(* CoDeSys 2.3.8.0 project: Laser_G67HP_3.pro *)
(* Libraries: STANDARD.LIB 5.6.98 12:03:02, TcBase.lib 6.6.06 16:41:28, TcSystem.lib 9.3.07 18:11:38, TcSystemCX.lib 5.3.07 17:55:46, TcUtilities.lib 29.3.07 15:04:14 *)

(* Global variable list: Globale_Variablen *)
VAR_GLOBAL

	(* Hardwareeingänge *)
	INot_Aus 			 	AT %IX0.0 : BOOL; (* Eingang 1 *)
	IDruckW			  	AT %IX0.1 : BOOL; (* Eingang 2 *)
	ISchututuer	  		AT %IX0.2 : BOOL; (* Eingang 3 *)
	ISchutzhaube  		AT %IX0.3 : BOOL; (* Eingang 4 *)
	IHWT_EIN			 	AT %IX0.4 : BOOL; (* Eingang 5 *)
	IHWT_AUS			AT %IX0.5 : BOOL; (* Eingang 6 *)
	IHWT_Quitt  			AT %IX0.6 : BOOL; (* Eingang 7 *)
	IRES1					AT %IX0.7 : BOOL; (* Eingang 8 *)

       IINI_Ueberlast  		AT %IX1.0 : BOOL; (* Eingang 9 *)
	IINI_IndexVor	  		AT %IX1.1 : BOOL; (* Eingang 10 *)
	IINI_IndexRueck  		AT %IX1.2 : BOOL; (* Eingang 11 *)
	IINI_Kupplung  		AT %IX1.3 : BOOL; (* Eingang 12 *)
	IINI_SpeicherZu		AT %IX1.4 : BOOL; (* Eingang 13 *)
	IRES3		 			AT %IX1.5 : BOOL; (* Eingang 14 *)
	IRES4					AT %IX1.6 : BOOL;
	IRES5		 			AT %IX1.7 : BOOL;

	IKammError  			AT %IX2.0 : BOOL; (* Eingang 17 *)
	IKammEnable  		AT %IX2.1 : BOOL; (* Eingang 18 *)
	IKammOutput  		AT %IX2.2 : BOOL; (* Eingang 19 *)
	IRES6		 			AT %IX2.3 : BOOL; (* Eingang 20 *)
	IAbsaug100P 			AT %IX2.4 : BOOL; (* Eingang 21 *)
	IAbsaugFilter			AT %IX2.5 : BOOL; (* Eingang 22 *)
	IRES					AT %IX2.6 : BOOL; (* Eingang 23 *)
	IFU_BB				AT %IX2.7 : BOOL; (* Eingang 24 *)

	IFrgMoma1 			AT %IX3.0 : BOOL;
	IFrgMoma2 			AT %IX3.1 : BOOL;
	ShutterZu	 			AT %IX3.2 : BOOL;
	ShutterAuf	 			AT %IX3.3 : BOOL;
	ILAS_HWFehler		AT %IX3.4 : BOOL;
	ILAS_SWIO 			AT %IX3.5 : BOOL;
	ILAS_Redy	 		AT %IX3.6 : BOOL;
	ILAS_AuftragEnde 	AT %IX3.7 : BOOL;

	ILasDataBit0 			AT %IX4.0 : BOOL;
	ILasDataBit1 	 		AT %IX4.1 : BOOL;
	ILasDataBit2 		 	AT %IX4.2 : BOOL;
	ILasDataBit3 		 	AT %IX4.3 : BOOL;
	ILasDataBit4 	 		AT %IX4.4 : BOOL;
	ILasDataBit5 	 		AT %IX4.5 : BOOL;
	ILasResI1	 		 	AT %IX4.6 : BOOL;
	ILasResI2 			 AT %IX4.7 : BOOL;

	(*Eingänge für die Panel Tasten*)

	IAPosKS1Input  		AT%IW20:INT;	 	(*Speicher 1 Füllstand analoger Eingang*)
	IARES1				AT%IW22:INT;
	IASSIDgInput			 AT %ID44:UDINT;	(* Drehgeber *)


	QHAmpelGn		 	AT %QX0.0 : BOOL; (* Ventil Pneumatik  *)
	QHAmpelRt	  		AT %QX0.1 : BOOL; (* Ausgang 2 *)
	QHAmpelGb 			AT %QX0.2 : BOOL; (* Ausgang 3 *)
	QRES1				AT %QX0.3 : BOOL; (* Ausgang 4 *)
	QHTasteEin			AT %QX0.4 : BOOL; (* Ausgang 5 *)
	QHTasteAus			AT %QX0.5 : BOOL; (* Ausgang 6 *)
	QHTasteQuitt			AT %QX0.6 : BOOL; (* Ausgang 7 *)
	QRES2				AT %QX0.7 : BOOL; (* Ausgang 8 *)

	QLasMark				AT %QX1.0 : BOOL; (* Ausgang 9 *)
	QLasMarkstop		AT %QX1.1 : BOOL; (* Ausgang 10 *)
	QLasProg1			AT %QX1.2 : BOOL; (* Ausgang 11 *)
	QLasProg2			AT %QX1.3 : BOOL; (* Ausgang 12 *)
	QLasRes2			AT %QX1.4 : BOOL; (* Ausgang 13 *)
	QLasRes3			AT %QX1.5 : BOOL; (* Ausgang 14 *)
	QFrgNaechst			AT %QX1.6 : BOOL; (* Ausgang 15 *)
	QAntriebeEin		     	AT %QX1.7 : BOOL; (* Ausgang 16 *)

	QMotVor	 			AT %QX2.0 : BOOL; (* Ausgang 9 *)
	QMotRueck			AT %QX2.1 : BOOL; (* Ausgang 10 *)
	QSaugAnford			AT %QX2.2 : BOOL; (* Ausgang 11 *)
	QVIndex				AT %QX2.3 : BOOL; (* Ausgang 12 *)
	QVUeberlast			AT %QX2.4 : BOOL; (* Ausgang 13 *)
	QVHaupt				AT %QX2.5 : BOOL; (* Ausgang 14 *)
	QVASpeicher			AT %QX2.6 : BOOL; (* Ausgang 15 *)
	QKammTrigg			AT %QX2.7 : BOOL; (* Ausgang 16 *)

	QASollwMot			AT%QW4:WORD; (*Ausgangswort 1*)
	QARes				 	AT%QW6:WORD; (*Ausgangswort 2*)

(* Anfang der Variablen für Kopmunikation SPS <> Visu *)
	TP_LaserAktiv	:			BOOL:= TRUE;
	TP_LaserHand:			BOOL;
	TP_RefSetzen:			BOOL;
	TP_KammeraAktiv:		BOOL:=TRUE;
	TP_MVor:					BOOL;
	TP_Mrueck:				BOOL;
	TP_MVorS:				BOOL;
	TP_MrueckS:				BOOL;

	TP_Hand:					BOOL;
	TP_Auto:					BOOL;
	TP_ZNullen:				BOOL;
	TPTypIndex:				WORD;
	TPTypSpeichern:			BOOL;
	TPKettenTyp: 				ARRAY[0..3] OF WORD;

	S_StUeberlast:			BOOL;
	S_StLaser:				BOOL;
	S_StKammera:			BOOL;
	S_StKupplung	:			BOOL;
	S_StSpeicherSchutz:		BOOL;
	S_StLaserSchutz:			BOOL;
	S_StSpeicher:				BOOL;
	S_StSammelstoerung:	BOOL;
	S_StDruck:				BOOL;
	S_StNotAus:				BOOL;
	S_StRef:					BOOL;
	S_StSchutzTuer:			BOOL;
	S_StSchutzhaube: 		BOOL;
	S_StAbsaugFilter:			BOOL;	(*Absauger Filter NIO*)
	S_StAbsaug100p:			BOOL;	(*Störung Absauger*)
	S_StShutter:				BOOL;

	S_StLasAuftragEnde:		BOOL;	(* Auftrag Ende*)
	S_StLasShutterZu:			BOOL;	(* Shutter zu *)
	S_StLasSoftware:			BOOL;	(*Software NIO*)
	S_StLasHardware:		BOOL;	(*Hardware NIO*)
	S_StIndexVor:			BOOL;	(*Index vor NIO*)
	S_StIndexRueck:			BOOL;	(*Index rueck NIO*)

	S_MSpeicherVoll:			BOOL;
	S_MShutterBetrieb:		BOOL;
	S_MSpeicherLeer:		BOOL;
	S_MWarteSpeicher:		BOOL;
	S_MHand:					BOOL;
	S_FKamera:				BOOL;
	S_FLaser:					BOOL;
	S_MAutoStart:				BOOL;
	S_MAutoStop:				BOOL;
	SI_Gliederzahl:			INT;
	SI_ProgNr:				INT;
	SI_FPosLaser:			INT;  (*wird nicht genutzt*)
	SI_FPosKamera:			INT;  (*wird nicht genutzt*)
	SKettenTyp:ARRAY[0..3] OF WORD;
(* ENDE*)

	Skal_IC_SSI_DG_Input: 	DINT;
	Skal_SSI_DG_4:			DINT;
	ZeigerReg:				INT;
	ZeigerKette: 				WORD;
	ImpulsPos: 				BOOL;
	ImpulsNeg: 				BOOL;
	Sammelstoerung: BOOL;

	V_Erster_Zyklus: BOOL;
	REF_IO: BOOL;
	AktTypIndexAlt: WORD;
	AktTypindex:WORD;
	NextTypIndex:WORD;
	PosErreicht: BOOL;


	NextTypIndexAlt: WORD;
	A_wechsell: BOOL;
	S1_AutoStop: BOOL;
	S2_Posstart: BOOL;
	S3_POSStop: BOOL;
	S4_IndexVor: BOOL;
	S5_LaserStart: BOOL;
	S6_IndexRueck: BOOL;

	Stoerunganlage:WORD;

	Zeiger_LMKontrolle: INT;
	FNichtMarkiert: BOOL;

	AktTypOL: BOOL;
	S_FrgEinzug: BOOL;
	KSEnIn: BOOL;
	KSEnOut: BOOL;
	TON_IIndexVor: TON;
	Stufe1: INT;
END_VAR

VAR_GLOBAL RETAIN



	(*Hinterlegte Kettentypen 64 Kettentypen 0-63  , 0=>Gliederzahl, 1-3=>Positionen der ersten bis dritten Außenlasche zum Lasern*)
	(*KettenTyp[x,2]=0 Bedeutet keine zweite Laserung an einer Kette*)
	(*KettenTyp[x,3]=0 Bedeutet keine dritte Laserung an einer Kette*)
	(*KettenTyp[x,1]=0 Nullter Kettentyp keine Laserung*)
	(*KettenTyp[x,0]=0 Ungültiger Eintrag *)

	(*Beispiel für eine Kette: 124 Glieder mit einer Laserung an der ersten Außenlasche gespeichert als Typ 5*)
	(*KettenTyp[5,0]=124   Kettentyp[5,1]=1 Kettentyp[5,2]=0  Kettentyp[5,3]=0*)
	KettenTyp							AT%QW100:ARRAY [0..63,0..3] OF WORD;

	(* Einträge in das Register RegMarkierung:
		X.0=1   Trennstelle
		X.1=1   Lasersollstelle, 
		X.2=1   Rückmeldung von Laser gelasert, 
		X.3=1   Fehler keine Rückmeldung von Laser "Gelesert"
		X.4=1   Rückmeldung Kammera Laserstelle
		X.5=1	Fehler keine Rückmeldung von Kammera "Laserstelle"
*)
	RegMarkierung					AT%QB1000:ARRAY[1..500] OF BYTE;


(*   Fehlerzähler für die erste Seite. Fehler können ohne Password zurückgesetzt werden*)

	SI_FKamera				AT%QW70:INT;
	SI_FLaser 				AT%QW72:INT;
	SI_IO						AT%QW74:INT;
	SI_NIO 					AT%QW76:INT;
(*	ZeigerGlied				AT%QW304:INT;				(* Zeiger für die Glieder in der Anlage zeigt auf das Glied unter der Trennstelle *)
	ZeigerAchtelGlied			AT%QW306:INT;
*)
END_VAR

(* Data type *)
TYPE DriveControl :
STRUCT
	ManOn: BOOL := FALSE; (* Visu -> SPS: Antrieb ein (nur bei FU-Antrieben) *)
	ManOff: BOOL := FALSE; (* Visu -> SPS: Antrieb aus (nur bei FU-Antrieben) *)
	ManFwd: BOOL := FALSE; (* Visu -> SPS: Antrieb im Handbetrieb langsam vorwärts *)
	ManBwd: BOOL := FALSE; (* Visu -> SPS: Antrieb im Handbetrieb langsam rückwärts *)
	TeilungVor: BOOL := FALSE; (* Visu -> SPS: Kette um eine Teilung vor (nur bei Servo-Antrieben) *)
	TeilungZur: BOOL := FALSE; (* Visu -> SPS: Kette um eine Teilung zurück (nur bei Servo-Antrieben) *)
	EnManCtrl: BOOL := FALSE; (* SPS -> Visu: Freigabe manuelle Steuerung *)
	ActOn: BOOL := FALSE; (* SPS -> Visu: Antrieb eingeschaltet *)
	ActOff: BOOL := FALSE; (* SPS -> Visu: Antrieb ausgeschaltet *)
	Error: BOOL := FALSE; (* SPS -> Visu: Störung Antrieb *)
END_STRUCT
END_TYPE

(* Data type *)
TYPE KettenTyp :
STRUCT
	PF: ARRAY [0..19] OF UDINT := 0,410,819,1229,1638,2048,2458,2867,3277,3686,4049,4506,4915,5328,5734,6144,6554,6963,7373,7782;

END_STRUCT
END_TYPE

(* Data type *)
TYPE KS_Control :
STRUCT
	EnInput: BOOL := FALSE; (* Freigabe Befüllen *)
	EnOutput: BOOL := FALSE; (* Freigabe Entleeren *)
	ActState: INT := 0; (* aktueller zustand für Visu *)
END_STRUCT
END_TYPE

(* Data type *)
TYPE KS_Control_1 :
STRUCT
	EnInput: BOOL := FALSE; (* Freigabe Befüllen *)
	EnOutput: BOOL := FALSE; (* Freigabe Entleeren *)
	ActState: INT := 0; (* aktueller zustand für Visu *)
END_STRUCT
END_TYPE

(* Data type *)
TYPE MotorControl :
STRUCT
	ManOn: BOOL := FALSE; (* Visu -> SPS: Antrieb im Handbetrieb ein *)
	ManOff: BOOL := FALSE; (* Visu -> SPS: Antrieb im Handbetrieb aus *)
	EnManCtrl: BOOL := FALSE; (* SPS -> Visu: Freigabe manuelle Steuerung *)
	ActOn: BOOL := FALSE; (* SPS -> Visu: Antrieb eingeschaltet *)
	ActOff: BOOL := FALSE; (* SPS -> Visu: Antrieb ausgeschaltet *)
	Error: BOOL := FALSE; (* SPS -> Visu: Störung Antrieb *)
END_STRUCT
END_TYPE

(* Data type *)
TYPE PneumControl :
STRUCT
	SetOn: BOOL := FALSE; (* Visu -> SPS: Arbeitsstellung anfahren *)
	SetOff: BOOL := FALSE; (* Visu -> SPS: Grundstellung anfahren *)
	EnSet: BOOL := FALSE; (* SPS -> Visu: Freigabe manuell Steuerung *)
	ActOn: BOOL := FALSE; (* SPS -> Visu: Zylinder in Arbeitsstellung *)
	ActOff: BOOL := FALSE; (* SPS -> Visu: Zylinder in Grundstellung *)
	Error: BOOL := FALSE; (* SPS -> Visu: Störung Zylinder oder Endschalter *)
END_STRUCT
END_TYPE

(* Data type *)
TYPE PosControl :
STRUCT
	PosSet: INT := 0; (* Positionssollwert [mm] *)
	ActPos: INT := 0; (* Positionsistwert [mm] *)
	PosLimitLo: INT := 0; (* unterer Grenzwert Sollposition [mm] *)
	PosLimitHi: INT := 0; (* oberer Grenzwert Sollposition [mm] *)
	StartPos: BOOL := FALSE; (* Visu -> SPS: Positionierung starten *)
	StoppPos: BOOL := FALSE; (* Visu -> SPS: Positionierung abbrechen *)
	ManPosUp: BOOL := FALSE; (* Visu -> SPS: Handbetrieb Positon erhöhen *)
	ManPosDn: BOOL := FALSE; (* Visu -> SPS: Handbetrieb Positon verringern *)
	EnPosSet: BOOL := FALSE; (* SPS -> Visu: Freigabe Sollwerteingabe *)
	EnManPos: BOOL := FALSE; (* SPS -> Visu: Freigabe manuelle Positionierung *)
	ActOn: BOOL := FALSE; (* SPS -> Visu: Antrieb eingeschaltet *)
	ActOff: BOOL := FALSE; (* SPS -> Visu: Antrieb ausgeschaltet *)
	Error: BOOL := FALSE; (* SPS -> Visu: Störung Antrieb *)
END_STRUCT
END_TYPE

(* Data type *)
TYPE StationControl :
STRUCT
	StepCounter: INT; (* SPS -> Visu: Schrittzähler *)
	SingleStep: BOOL := FALSE; (* Visu -> SPS: Einzelschritt weiterschalten *)
	SingleCycle: BOOL := FALSE; (* Visu -> SPS: Einzelzyklus ausführen *)
	StartCycle: BOOL := FALSE; (* Zyklus im Auto-Betrieb starten *)
	ManInit: BOOL := FALSE; (* Visu -> SPS: Grundstellung anfahren *)
	AutoInit: BOOL := FALSE; (* Grundstellung im Auto-Betrieb anfahren *)
	SetFinished: BOOL := FALSE; (* Visu -> SPS: Fertigmeldung setzen *)
	WaitPos: BOOL := FALSE; (* Station in Warteposition für Stopp *)
	EnSemiAutoCtrl: BOOL := FALSE; (* SPS -> Visu: Steuerung Halbautomatikbetrieb freigeben; Freigabe für SingleStep, SingleCycle, InitPos und SetFinished *)
	InitPos: BOOL := FALSE; (* Station in Grundstellung *)
	Finished: BOOL := FALSE; (* Station fertig *)
	ErrorInitPos: BOOL := FALSE; (* Störung Grundstellung nicht erreicht *)
	ErrorCycleTime: BOOL := FALSE; (* Störung Zeitüberschreitung Zyklus *)
	ActState: INT := 0; (* SPS -> Visu: Zustand der Station: 0 = Störung, 1 = bereit, 2 = aktiv *)
END_STRUCT
END_TYPE

(* POU INIT, ST *)
PROGRAM INIT

VAR

END_VAR
(* Der Kettentyp wird von Laserrechner ausgewählt *)
NextTypIndex.0:=ILasDataBit0;
NextTypIndex.1:=ILasDataBit1;
NextTypIndex.2:=ILasDataBit2;
NextTypIndex.3:=ILasDataBit3;
NextTypIndex.4:=ILasDataBit4;
NextTypIndex.5:=ILasDataBit5;



(*  Wenn NuxtTypIndex = 0 dann Auftrag ohne Laserung *)
(* Wenn Laser per Touchpannel deaktiviert dann auch Auftrag ohne Laserung *)
IF TP_LaserAktiv = FALSE THEN
	NextTypIndex:=0;
END_IF

(* Wenn Wechsell von Auftrag ohne Laserung auf Auftrag mit Laserung dann Referenz nue anfordern *)

IF	AktTypIndex = 0 AND NextTypIndex <> 0 THEN
	REF_IO:=FALSE;
END_IF




(* Wenn die Maschine eingeschaltet wird ist eine Ref Fahrt durchzuführen *)
IF V_Erster_Zyklus=FALSE THEN
	REF_IO:=FALSE;
	AktTypIndex:=NextTypIndex;
END_IF
V_Erster_Zyklus:=TRUE;



(* Trennstelle der Kette auf Indexposition fahren und Referenzieren *)
IF (*REF_IO= FALSE AND*) TP_RefSetzen= TRUE THEN
	ZeigerKette:=KettenTyp[AktTypIndex,0];
	REF_IO:=TRUE;
END_IF


(* Wenn Kettentyp gewechselt wurde muß Auftragswechsellbitt gesetzt werden *)
IF NextTypIndex <> NextTypIndexAlt THEN
	A_wechsell:=TRUE;
END_IF
NextTypIndexAlt:=NextTypIndex;

(* Der Auftragswechsell wird durchgeführt wenn das Ende der  Kette von Alten Auftrag unter der Leserstelle gelangt *)
(* Auftragswechsellbit wird auf FALSE gesetzt *)
IF   ZeigerKette = KettenTyp[AktTypIndex,0] THEN
	AktTypIndex:=NextTypIndex;
	SI_ProgNr:=AktTypIndex;
	SI_Gliederzahl:= KettenTyp[AktTypIndex,0];
	A_wechsell:=FALSE;
	ZeigerKette := KettenTyp[AktTypIndex,0];
END_IF

IF	NextTypIndex = 63 THEN
	SI_ProgNr:=63;
END_IF

IF	ImpulsPos =TRUE THEN
	(*Alten Eintrag im Register Löschen*)
	(*Laser wird dann die Markierung eintragen*)
	RegMarkierung[ZeigerReg]:=0;

	(*Trennstell in das Register eintragen*)
	IF   ZeigerKette = KettenTyp[AktTypIndex,0] THEN
	RegMarkierung[ZeigerReg].0:=TRUE;
	END_IF

END_IF
END_PROGRAM

(* POU MAIN_1, FBD *)
PROGRAM MAIN_1
VAR
	SollPos1: SollPos;
	ASMSollW1: AsmSollW;
	Motorsteuerung1: Motorsteuerun;
	Betriebsarten1: Betriebsarten;
	Kettenspeicher1: Kettenspeicher;

	Saugersteuerung1: Saugersteuerung;
	Kettentypen1: Kettentypen;
	Indexsteuerung1: Indexsteuernung;
	Anlagenstoerung1: Anlagestoerung;
	Lasersteuerung1: Lasersteuerung;
	LaserMeldungKontrolle1: LaserMeldungKontrolle;
	Kammera1: Kammera;
	FK1: BOOL;
	V1: BOOL;
	PF1: R_TRIG;
	TP1: TP;
END_VAR
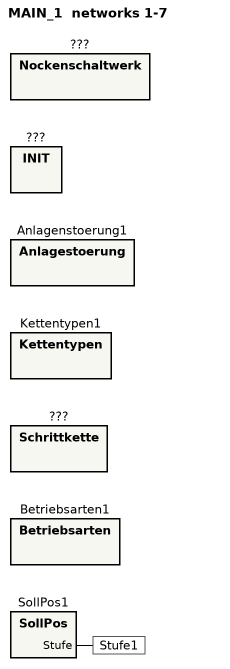
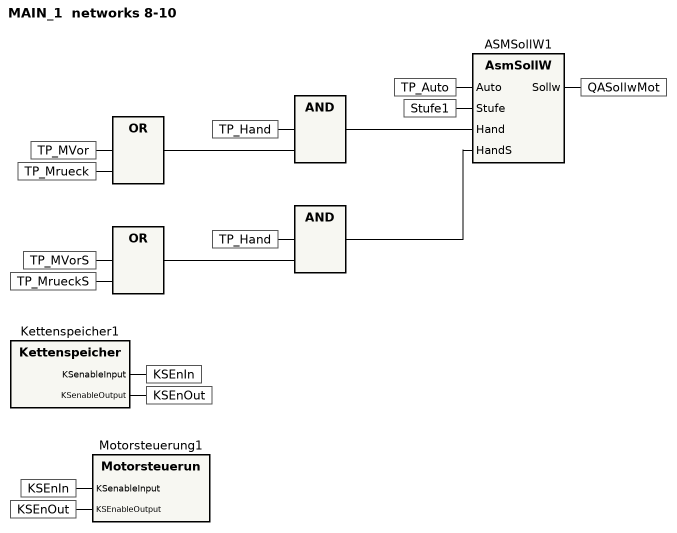
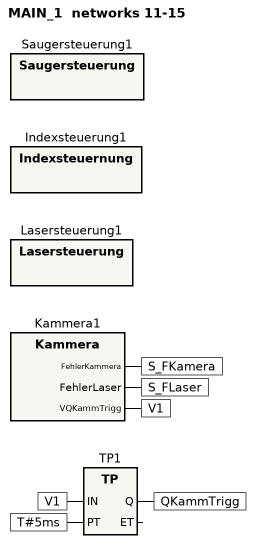
_FBD_ (* Function Block Diagram *)
NETWORK 1
	???:Nockenschaltwerk()
NETWORK 2
	???:INIT()
NETWORK 3
	Anlagenstoerung1:Anlagestoerung()
NETWORK 4
	Kettentypen1:Kettentypen()
NETWORK 5
	???:Schrittkette()
NETWORK 6
	Betriebsarten1:Betriebsarten()
NETWORK 7
	SollPos1:SollPos() => Stufe1
NETWORK 8
	ASMSollW1:AsmSollW(Auto: TP_Auto, Stufe: Stufe1, Hand: AND(TP_Hand, OR(TP_MVor, TP_Mrueck)), HandS: AND(TP_Hand, OR(TP_MVorS, TP_MrueckS))) => QASollwMot
NETWORK 9
	Kettenspeicher1:Kettenspeicher(KSenableOutput => KSEnOut) => KSEnIn
NETWORK 10
	Motorsteuerung1:Motorsteuerun(KSenableInput: KSEnIn, KSEnableOutput: KSEnOut)
NETWORK 11
	Saugersteuerung1:Saugersteuerung()
NETWORK 12
	Indexsteuerung1:Indexsteuernung()
NETWORK 13
	Lasersteuerung1:Lasersteuerung()
NETWORK 14
	Kammera1:Kammera(FehlerLaser => S_FLaser, VQKammTrigg => V1) => S_FKamera
NETWORK 15
	TP1:TP(IN: V1, PT: T#5ms) => QKammTrigg
_END_FBD_
(* the same logic as Structured Text *)
(* Network 1: see the listing above *)
(* Network 2: see the listing above *)
(* Network 3 *)
Anlagenstoerung1();
(* Network 4 *)
Kettentypen1();
(* Network 5: see the listing above *)
(* Network 6 *)
Betriebsarten1();
(* Network 7 *)
SollPos1();
Stufe1 := SollPos1.Stufe;
(* Network 8 *)
ASMSollW1(Auto := TP_Auto, Stufe := Stufe1, Hand := TP_Hand AND (TP_MVor OR TP_Mrueck), HandS := TP_Hand AND (TP_MVorS OR TP_MrueckS));
QASollwMot := ASMSollW1.Sollw;
(* Network 9 *)
Kettenspeicher1();
KSEnOut := Kettenspeicher1.KSenableOutput;
KSEnIn := Kettenspeicher1.KSenableInput;
(* Network 10 *)
Motorsteuerung1(KSenableInput := KSEnIn, KSEnableOutput := KSEnOut);
(* Network 11 *)
Saugersteuerung1();
(* Network 12 *)
Indexsteuerung1();
(* Network 13 *)
Lasersteuerung1();
(* Network 14 *)
Kammera1();
S_FLaser := Kammera1.FehlerLaser;
V1 := Kammera1.VQKammTrigg;
S_FKamera := Kammera1.FehlerKammera;
(* Network 15 *)
TP1(IN := V1, PT := T#5ms);
QKammTrigg := TP1.Q;
END_PROGRAM

(* POU Funktionsbausteine/SollPos, ST *)
FUNCTION_BLOCK SollPos
VAR_INPUT
END_VAR
VAR_OUTPUT
	Stufe: INT := 1;
END_VAR
VAR
	ZeigerStufe1: INT;
	ZeigerStufe2: INT;
	ZeigerStufe3: INT;
	ZeigerStufe4: INT;
	ZeigerStufe5: INT;

END_VAR
(* Wenn Referenz gesetzt oder wurde oder nach dem Einschalten erst langsam anfahren *)

IF TP_RefSetzen= TRUE OR V_Erster_Zyklus= FALSE THEN
	Stufe:=1;
END_IF

 TP_RefSetzen:= FALSE;


IF	ImpulsPos =TRUE THEN


	(* Geschwindigkeitsstufen für die Positionierung ermitteln *)
	(* Zeiger für die Stufen berechnen *)
	(* Bearbeitung nur wenn Aussenlasche*)
	IF ZeigerKette.0=FALSE THEN
		ZeigerStufe1:=ZeigerKette+2;
		IF ZeigerStufe1>KettenTyp[AktTypindex,0] THEN
			ZeigerStufe1:=ZeigerStufe1-KettenTyp[AktTypindex,0];
		END_IF
		ZeigerStufe2:=ZeigerStufe1+2;
		IF ZeigerStufe2>KettenTyp[AktTypindex,0] THEN
			ZeigerStufe2:=ZeigerStufe2-KettenTyp[AktTypindex,0];
		END_IF
		ZeigerStufe3:=ZeigerStufe2+2;
		IF ZeigerStufe3>KettenTyp[AktTypindex,0] THEN
			ZeigerStufe3:=ZeigerStufe3-KettenTyp[AktTypindex,0];
		END_IF
		ZeigerStufe4:=ZeigerStufe3+2;
		IF ZeigerStufe4>KettenTyp[AktTypindex,0] THEN
			ZeigerStufe4:=ZeigerStufe4-KettenTyp[AktTypindex,0];
		END_IF
		ZeigerStufe5:=ZeigerStufe4+2;
		IF ZeigerStufe5>KettenTyp[AktTypindex,0] THEN
			ZeigerStufe5:=ZeigerStufe5-KettenTyp[AktTypindex,0];
		END_IF




		(* In Abhängikeit von der Entfernung der nächsten Lasche welche gelesert werden soll wird die Geschwindigkeit des Motors in 6 Stufen geregelt*)
		(* Wenn Auftragswechsell anliegt wird die Geschwindigkeit des Motors verringert bisdas Ende der alten Kette die Laserungsstelle erreicht*)
		(* Sollgeschwindigkeit ist auf Stufe 6 eingestellt. Wenn die Laserungsstelle auf fünfte Aussenlasche vor Laserungsstelle ist dann langsamer auf Stufe 5*)

		IF ZeigerStufe5 = KettenTyp[AktTypindex,1]*2 OR ZeigerStufe5 = KettenTyp[AktTypindex,2]*2 OR ZeigerStufe5 = KettenTyp[AktTypindex,3]*2THEN
			Stufe:=5;
		ELSE
			Stufe:=6;
		END_IF
		(* Wenn Auftragswechsell und Kettenende von alten Auftrag auf 5 Außenlasche vor Laserungsstelle dan auf Stufe 5 stellen*)
		IF	A_wechsell = TRUE AND (ZeigerKette+10) = KettenTyp[AktTypindex,0] THEN
			Stufe:=5;
		END_IF


		(* Wenn die Laserungsstelle auf vierte Aussenlasche vor Laserungsstelle ist dann langsamer auf Stufe 4*)
		IF ZeigerStufe4 = KettenTyp[AktTypindex,1]*2 OR ZeigerStufe4 = KettenTyp[AktTypindex,2]*2 OR ZeigerStufe4 = KettenTyp[AktTypindex,3]*2THEN
			Stufe:=4;
		END_IF
		(* Wenn Auftragswechsell und Kettenende von alten Auftrag auf 4 Außenlasche vor Laserungsstelle dan auf Stufe 4 stellen*)
		IF	A_wechsell = TRUE AND (ZeigerKette+8) = KettenTyp[AktTypindex,0] THEN
			Stufe:=4;
		END_IF



		IF ZeigerStufe3 = KettenTyp[AktTypindex,1]*2 OR ZeigerStufe3 = KettenTyp[AktTypindex,2]*2 OR ZeigerStufe3 = KettenTyp[AktTypindex,3]*2THEN
			Stufe:=3;
		END_IF
		(* Wenn Auftragswechsell und Kettenende von alten Auftrag auf 3 Außenlasche vor Laserungsstelle dan auf Stufe 3 stellen*)
		IF	A_wechsell = TRUE AND (ZeigerKette+6) = KettenTyp[AktTypindex,0] THEN
			Stufe:=3;
		END_IF



		IF ZeigerStufe2 = KettenTyp[AktTypindex,1]*2 OR ZeigerStufe2 = KettenTyp[AktTypindex,2]*2 OR ZeigerStufe2 = KettenTyp[AktTypindex,3]*2THEN
			Stufe:=2;
		END_IF
		(* Wenn Auftragswechsell und Kettenende von alten Auftrag auf 2 Außenlasche vor Laserungsstelle dan auf Stufe 2 stellen*)
		IF	A_wechsell = TRUE AND (ZeigerKette+4) = KettenTyp[AktTypindex,0] THEN
			Stufe:=2;
		END_IF

		IF ZeigerStufe1 = KettenTyp[AktTypindex,1]*2 OR ZeigerStufe1 = KettenTyp[AktTypindex,2]*2 OR ZeigerStufe1 = KettenTyp[AktTypindex,3]*2THEN
			Stufe:=1;
		END_IF
		(* Wenn Auftragswechsell und Kettenende von alten Auftrag auf 1 Außenlasche vor Laserungsstelle dan auf Stufe 1 stellen*)
		IF	A_wechsell = TRUE AND (ZeigerKette+2) = KettenTyp[AktTypindex,0] THEN
			Stufe:=1;
		END_IF

		(* Position erreicht melden und Laserungssollstelle in das Register Schreiben *)
		IF ZeigerKette = KettenTyp[AktTypindex,1]*2 OR ZeigerKette = KettenTyp[AktTypindex,2]*2 OR ZeigerKette = KettenTyp[AktTypindex,3]*2THEN
			IF RegMarkierung[ZeigerReg].2 = FALSE THEN
				PosErreicht:=TRUE;
				RegMarkierung[ZeigerReg].1:=TRUE;
			END_IF
		END_IF
	END_IF


	(*  Bearbeitung nur bei Innenlasche an der Laserstelle *)
	(*  Wenn die Lasersollposition überfahren ohne zu lasern dann  PosErreicht zurücksetzen *)
	IF ZeigerKette.0=TRUE  THEN
	PosErreicht:=FALSE;
	END_IF

END_IF
END_FUNCTION_BLOCK

(* POU Funktionsbausteine/AsmSollW, ST *)
FUNCTION_BLOCK AsmSollW
VAR

END_VAR

VAR_INPUT
	Auto: BOOL;
	Stufe: INT;
	Hand: BOOL;
	HandS:BOOL;
END_VAR
VAR_OUTPUT
	Sollw: INT;
END_VAR
IF  Auto = TRUE THEN
	IF Stufe= 6 THEN
	Sollw:=30000;
	END_IF
	IF Stufe= 5 THEN
	Sollw:=27000;
	END_IF
	IF Stufe= 4 THEN
	Sollw:=18000;
	END_IF
	IF Stufe= 3 THEN
	Sollw:=15000;
	END_IF
	IF Stufe= 2 THEN
	Sollw:=10000;
	END_IF
	IF Stufe= 1 THEN
	Sollw:=1000;
	END_IF
END_IF

IF	Hand=TRUE  THEN
	Sollw:=5000;
END_IF


IF	HandS=TRUE  THEN
	Sollw:=15000;
END_IF
END_FUNCTION_BLOCK

(* POU Funktionsbausteine/Motorsteuerun, FBD *)
FUNCTION_BLOCK Motorsteuerun
VAR_INPUT
	KSenableInput: BOOL;
	KSEnableOutput: BOOL;
END_VAR
VAR_OUTPUT
END_VAR
VAR
	PF_AutoStart: R_TRIG;
	PF_AutoStop: R_TRIG;
	StopGoMot: RS;
END_VAR
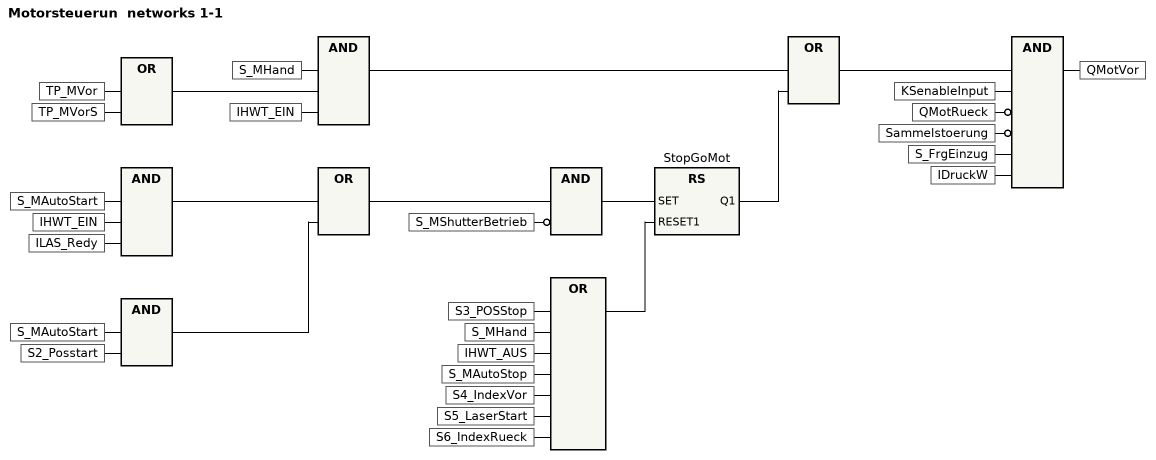
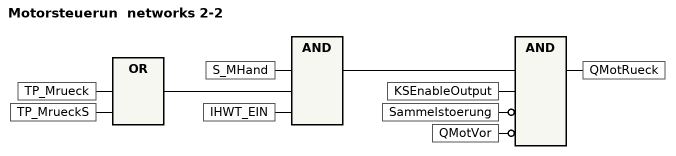
_FBD_ (* Function Block Diagram *)
NETWORK 1 (* Ansteuerung des Motors M1 in Positive richtung *)
	AND(OR(AND(S_MHand, OR(TP_MVor, TP_MVorS), IHWT_EIN), StopGoMot:RS(SET: AND(OR(AND(S_MAutoStart, IHWT_EIN, ILAS_Redy), AND(S_MAutoStart, S2_Posstart)), NOT S_MShutterBetrieb), RESET1: OR(S3_POSStop, S_MHand, IHWT_AUS, S_MAutoStop, S4_IndexVor, S5_LaserStart, S6_IndexRueck))), KSenableInput, NOT QMotRueck, NOT Sammelstoerung, S_FrgEinzug, IDruckW) => QMotVor
NETWORK 2 (* Ansteuerung Motor M1 in negative Richtung *)
	AND(AND(S_MHand, OR(TP_Mrueck, TP_MrueckS), IHWT_EIN), KSEnableOutput, NOT Sammelstoerung, NOT QMotVor) => QMotRueck
_END_FBD_
(* the same logic as Structured Text *)
(* Network 1: Ansteuerung des Motors M1 in Positive richtung *)
StopGoMot(SET := ((S_MAutoStart AND IHWT_EIN AND ILAS_Redy) OR (S_MAutoStart AND S2_Posstart)) AND NOT S_MShutterBetrieb, RESET1 := S3_POSStop OR S_MHand OR IHWT_AUS OR S_MAutoStop OR S4_IndexVor OR S5_LaserStart OR S6_IndexRueck);
QMotVor := ((S_MHand AND (TP_MVor OR TP_MVorS) AND IHWT_EIN) OR StopGoMot.Q1) AND KSenableInput AND NOT QMotRueck AND NOT Sammelstoerung AND S_FrgEinzug AND IDruckW;
(* Network 2: Ansteuerung Motor M1 in negative Richtung *)
QMotRueck := (S_MHand AND (TP_Mrueck OR TP_MrueckS) AND IHWT_EIN) AND KSEnableOutput AND NOT Sammelstoerung AND NOT QMotVor;
END_FUNCTION_BLOCK

(* POU Funktionsbausteine/Betriebsarten, FBD *)
FUNCTION_BLOCK Betriebsarten
VAR_INPUT
END_VAR
VAR_OUTPUT
END_VAR
VAR
	Blink_TON1: TON;
	Blink_TON2: TON;
	VIHWT_AUS: BOOL;
END_VAR
VAR (* helpers for the ST form of the networks *)
	_p1 : BOOL;
	_p2 : BOOL;
END_VAR
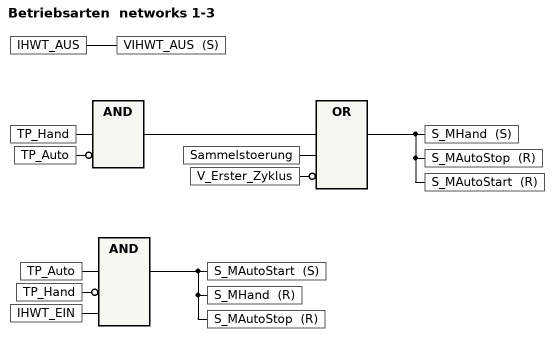
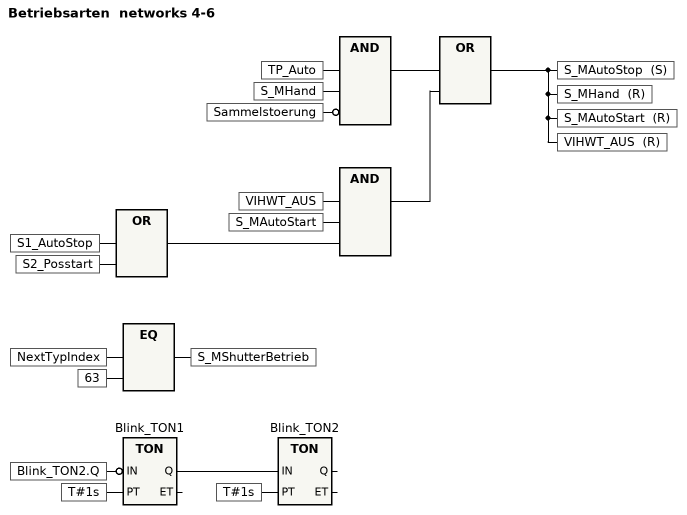
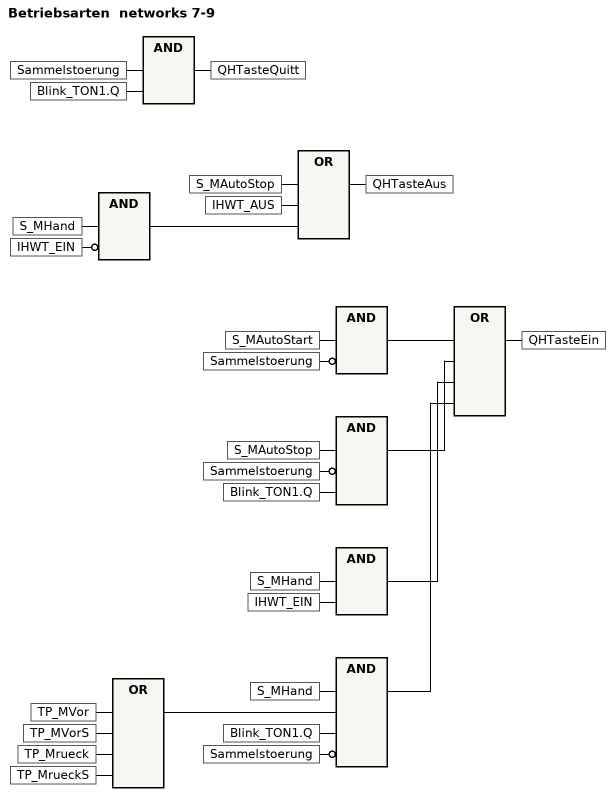
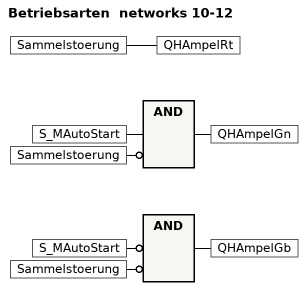
_FBD_ (* Function Block Diagram *)
NETWORK 1
	IHWT_AUS => S VIHWT_AUS
NETWORK 2
	OR(AND(TP_Hand, NOT TP_Auto), Sammelstoerung, NOT V_Erster_Zyklus) => S S_MHand, R S_MAutoStop, R S_MAutoStart
NETWORK 3
	AND(TP_Auto, NOT TP_Hand, IHWT_EIN) => S S_MAutoStart, R S_MHand, R S_MAutoStop
NETWORK 4
	OR(AND(TP_Auto, S_MHand, NOT Sammelstoerung), AND(VIHWT_AUS, S_MAutoStart, OR(S1_AutoStop, S2_Posstart))) => S S_MAutoStop, R S_MHand, R S_MAutoStart, R VIHWT_AUS
NETWORK 5
	EQ(NextTypIndex, 63) => S_MShutterBetrieb
NETWORK 6
	Blink_TON2:TON(IN: Blink_TON1:TON(IN: NOT Blink_TON2.Q, PT: T#1s), PT: T#1s)
NETWORK 7
	AND(Sammelstoerung, Blink_TON1.Q) => QHTasteQuitt
NETWORK 8
	OR(S_MAutoStop, IHWT_AUS, AND(S_MHand, NOT IHWT_EIN)) => QHTasteAus
NETWORK 9
	OR(AND(S_MAutoStart, NOT Sammelstoerung), AND(S_MAutoStop, NOT Sammelstoerung, Blink_TON1.Q), AND(S_MHand, IHWT_EIN), AND(S_MHand, OR(TP_MVor, TP_MVorS, TP_Mrueck, TP_MrueckS), Blink_TON1.Q, NOT Sammelstoerung)) => QHTasteEin
NETWORK 10
	Sammelstoerung => QHAmpelRt
NETWORK 11
	AND(S_MAutoStart, NOT Sammelstoerung) => QHAmpelGn
NETWORK 12
	AND(NOT S_MAutoStart, NOT Sammelstoerung) => QHAmpelGb
_END_FBD_
(* the same logic as Structured Text *)
(* Network 1 *)
IF IHWT_AUS THEN VIHWT_AUS := TRUE; END_IF;
(* Network 2 *)
_p1 := (TP_Hand AND NOT TP_Auto) OR Sammelstoerung OR NOT V_Erster_Zyklus;
IF _p1 THEN S_MHand := TRUE; S_MAutoStop := FALSE; S_MAutoStart := FALSE; END_IF;
(* Network 3 *)
IF TP_Auto AND NOT TP_Hand AND IHWT_EIN THEN S_MAutoStart := TRUE; S_MHand := FALSE; S_MAutoStop := FALSE; END_IF;
(* Network 4 *)
_p2 := (TP_Auto AND S_MHand AND NOT Sammelstoerung) OR (VIHWT_AUS AND S_MAutoStart AND (S1_AutoStop OR S2_Posstart));
IF _p2 THEN S_MAutoStop := TRUE; S_MHand := FALSE; S_MAutoStart := FALSE; VIHWT_AUS := FALSE; END_IF;
(* Network 5 *)
S_MShutterBetrieb := NextTypIndex = 63;
(* Network 6 *)
Blink_TON1(IN := NOT Blink_TON2.Q, PT := T#1s);
Blink_TON2(IN := Blink_TON1.Q, PT := T#1s);
(* Network 7 *)
QHTasteQuitt := Sammelstoerung AND Blink_TON1.Q;
(* Network 8 *)
QHTasteAus := S_MAutoStop OR IHWT_AUS OR (S_MHand AND NOT IHWT_EIN);
(* Network 9 *)
QHTasteEin := (S_MAutoStart AND NOT Sammelstoerung) OR (S_MAutoStop AND NOT Sammelstoerung AND Blink_TON1.Q) OR (S_MHand AND IHWT_EIN) OR (S_MHand AND (TP_MVor OR TP_MVorS OR TP_Mrueck OR TP_MrueckS) AND Blink_TON1.Q AND NOT Sammelstoerung);
(* Network 10 *)
QHAmpelRt := Sammelstoerung;
(* Network 11 *)
QHAmpelGn := S_MAutoStart AND NOT Sammelstoerung;
(* Network 12 *)
QHAmpelGb := NOT S_MAutoStart AND NOT Sammelstoerung;
END_FUNCTION_BLOCK

(* POU Funktionsbausteine/Kettenspeicher, FBD *)
FUNCTION_BLOCK Kettenspeicher
VAR_INPUT
END_VAR
VAR_OUTPUT
	KSenableInput: BOOL;
	KSenableOutput: BOOL;
END_VAR
VAR
	RS1: RS;
END_VAR
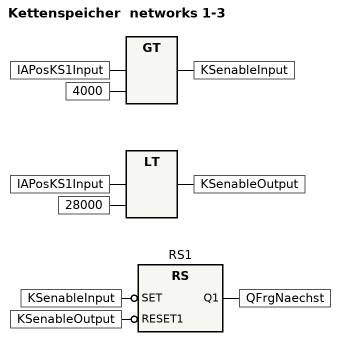
_FBD_ (* Function Block Diagram *)
NETWORK 1
	GT(IAPosKS1Input, 4000) => KSenableInput
NETWORK 2
	LT(IAPosKS1Input, 28000) => KSenableOutput
NETWORK 3
	RS1:RS(SET: NOT KSenableInput, RESET1: NOT KSenableOutput) => QFrgNaechst
_END_FBD_
(* the same logic as Structured Text *)
(* Network 1 *)
KSenableInput := IAPosKS1Input > 4000;
(* Network 2 *)
KSenableOutput := IAPosKS1Input < 28000;
(* Network 3 *)
RS1(SET := NOT KSenableInput, RESET1 := NOT KSenableOutput);
QFrgNaechst := RS1.Q1;
END_FUNCTION_BLOCK

(* POU Funktionsbausteine/Saugersteuerung, FBD *)
FUNCTION_BLOCK Saugersteuerung
VAR_INPUT
END_VAR
VAR_OUTPUT
END_VAR
VAR
	TON1: TON;
	TOF1: TOF;
END_VAR
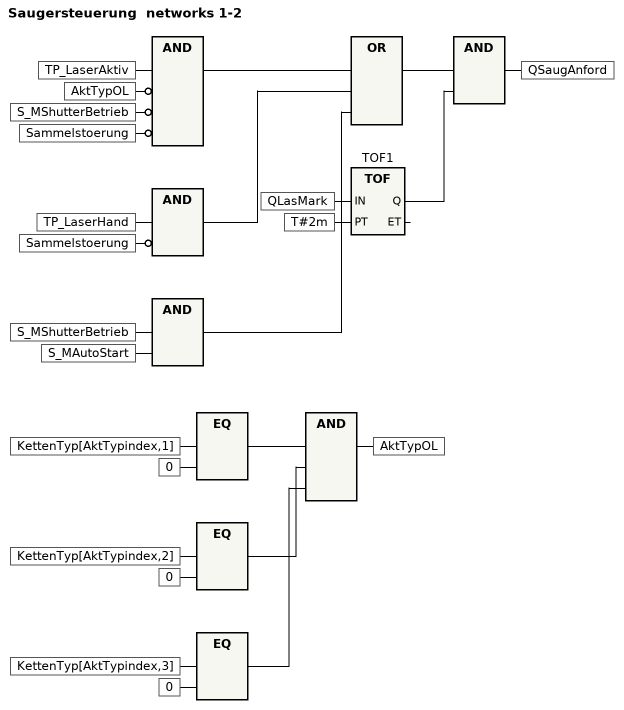
_FBD_ (* Function Block Diagram *)
NETWORK 1
	AND(OR(AND(TP_LaserAktiv, NOT AktTypOL, NOT S_MShutterBetrieb, NOT Sammelstoerung), AND(TP_LaserHand, NOT Sammelstoerung), AND(S_MShutterBetrieb, S_MAutoStart)), TOF1:TOF(IN: QLasMark, PT: T#2m)) => QSaugAnford
NETWORK 2
	AND(EQ(KettenTyp[AktTypindex,1], 0), EQ(KettenTyp[AktTypindex,2], 0), EQ(KettenTyp[AktTypindex,3], 0)) => AktTypOL
_END_FBD_
(* the same logic as Structured Text *)
(* Network 1 *)
TOF1(IN := QLasMark, PT := T#2m);
QSaugAnford := ((TP_LaserAktiv AND NOT AktTypOL AND NOT S_MShutterBetrieb AND NOT Sammelstoerung) OR (TP_LaserHand AND NOT Sammelstoerung) OR (S_MShutterBetrieb AND S_MAutoStart)) AND TOF1.Q;
(* Network 2 *)
AktTypOL := ((KettenTyp[AktTypindex,1]) = 0) AND ((KettenTyp[AktTypindex,2]) = 0) AND ((KettenTyp[AktTypindex,3]) = 0);
END_FUNCTION_BLOCK

(* POU Funktionsbausteine/Kettentypen, ST *)
FUNCTION_BLOCK Kettentypen
VAR_INPUT
END_VAR
VAR_OUTPUT
END_VAR
VAR
END_VAR
(*  Angewählten Kettentyp für Visu bereitstellen *)

SKettenTyp[0]:=KettenTyp[TPTypIndex,0];
SKettenTyp[1]:=KettenTyp[TPTypIndex,1];
SKettenTyp[2]:=KettenTyp[TPTypIndex,2];
SKettenTyp[3]:=KettenTyp[TPTypIndex,3];


(* Editierte Kettentypen remanent speichern *)
IF TPTypSpeichern = TRUE THEN
	KettenTyp[TPTypIndex,0]:=TPKettenTyp[0];
	KettenTyp[TPTypIndex,1]:=TPKettenTyp[1];
	KettenTyp[TPTypIndex,2]:=TPKettenTyp[2];
	KettenTyp[TPTypIndex,3]:=TPKettenTyp[3];
END_IF

TPTypSpeichern:= FALSE;
END_FUNCTION_BLOCK

(* POU Funktionsbausteine/Indexsteuernung, FBD *)
FUNCTION_BLOCK Indexsteuernung
VAR_INPUT
END_VAR
VAR_OUTPUT
END_VAR
VAR
	SR1: RS;
	PF_1: R_TRIG;
	PF2: R_TRIG;
	PF_3: R_TRIG;
	PF_4: R_TRIG;
	PF_5: R_TRIG;
END_VAR
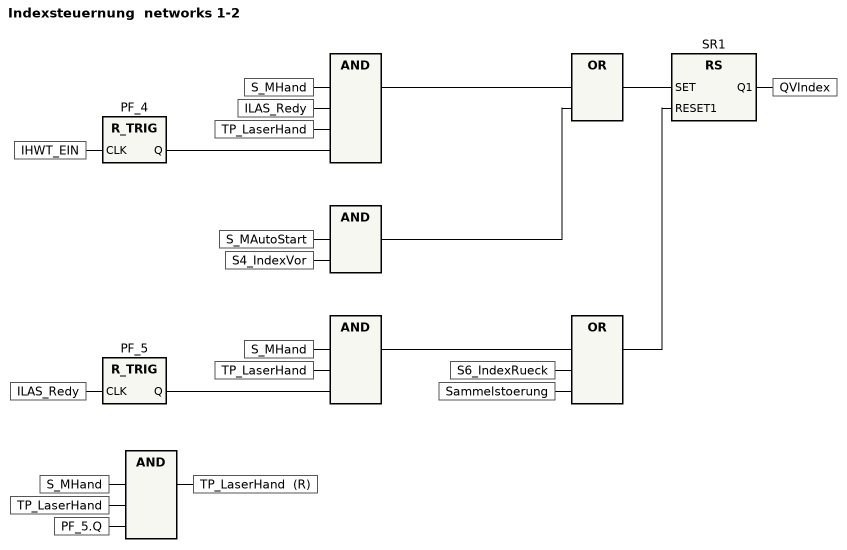
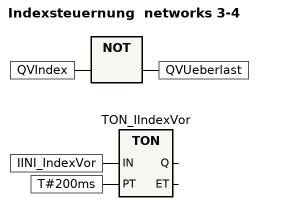
_FBD_ (* Function Block Diagram *)
NETWORK 1
	SR1:RS(SET: OR(AND(S_MHand, ILAS_Redy, TP_LaserHand, PF_4:R_TRIG(CLK: IHWT_EIN)), AND(S_MAutoStart, S4_IndexVor)), RESET1: OR(AND(S_MHand, TP_LaserHand, PF_5:R_TRIG(CLK: ILAS_Redy)), S6_IndexRueck, Sammelstoerung)) => QVIndex
NETWORK 2
	AND(S_MHand, TP_LaserHand, PF_5.Q) => R TP_LaserHand
NETWORK 3
	NOT QVIndex => QVUeberlast
NETWORK 4
	TON_IIndexVor:TON(IN: IINI_IndexVor, PT: T#200ms)
_END_FBD_
(* the same logic as Structured Text *)
(* Network 1 *)
PF_4(CLK := IHWT_EIN);
PF_5(CLK := ILAS_Redy);
SR1(SET := (S_MHand AND ILAS_Redy AND TP_LaserHand AND PF_4.Q) OR (S_MAutoStart AND S4_IndexVor), RESET1 := (S_MHand AND TP_LaserHand AND PF_5.Q) OR S6_IndexRueck OR Sammelstoerung);
QVIndex := SR1.Q1;
(* Network 2 *)
IF S_MHand AND TP_LaserHand AND PF_5.Q THEN TP_LaserHand := FALSE; END_IF;
(* Network 3 *)
QVUeberlast := NOT QVIndex;
(* Network 4 *)
TON_IIndexVor(IN := IINI_IndexVor, PT := T#200ms);
END_FUNCTION_BLOCK

(* POU Funktionsbausteine/Anlagestoerung, FBD *)
FUNCTION_BLOCK Anlagestoerung
VAR_INPUT
END_VAR
VAR_OUTPUT
END_VAR
VAR

	TON1: TON;
	PF_1: R_TRIG;
	TOF1: TOF;
	TON2: TON;
	TON3: TON;
	TON4: TON;
END_VAR
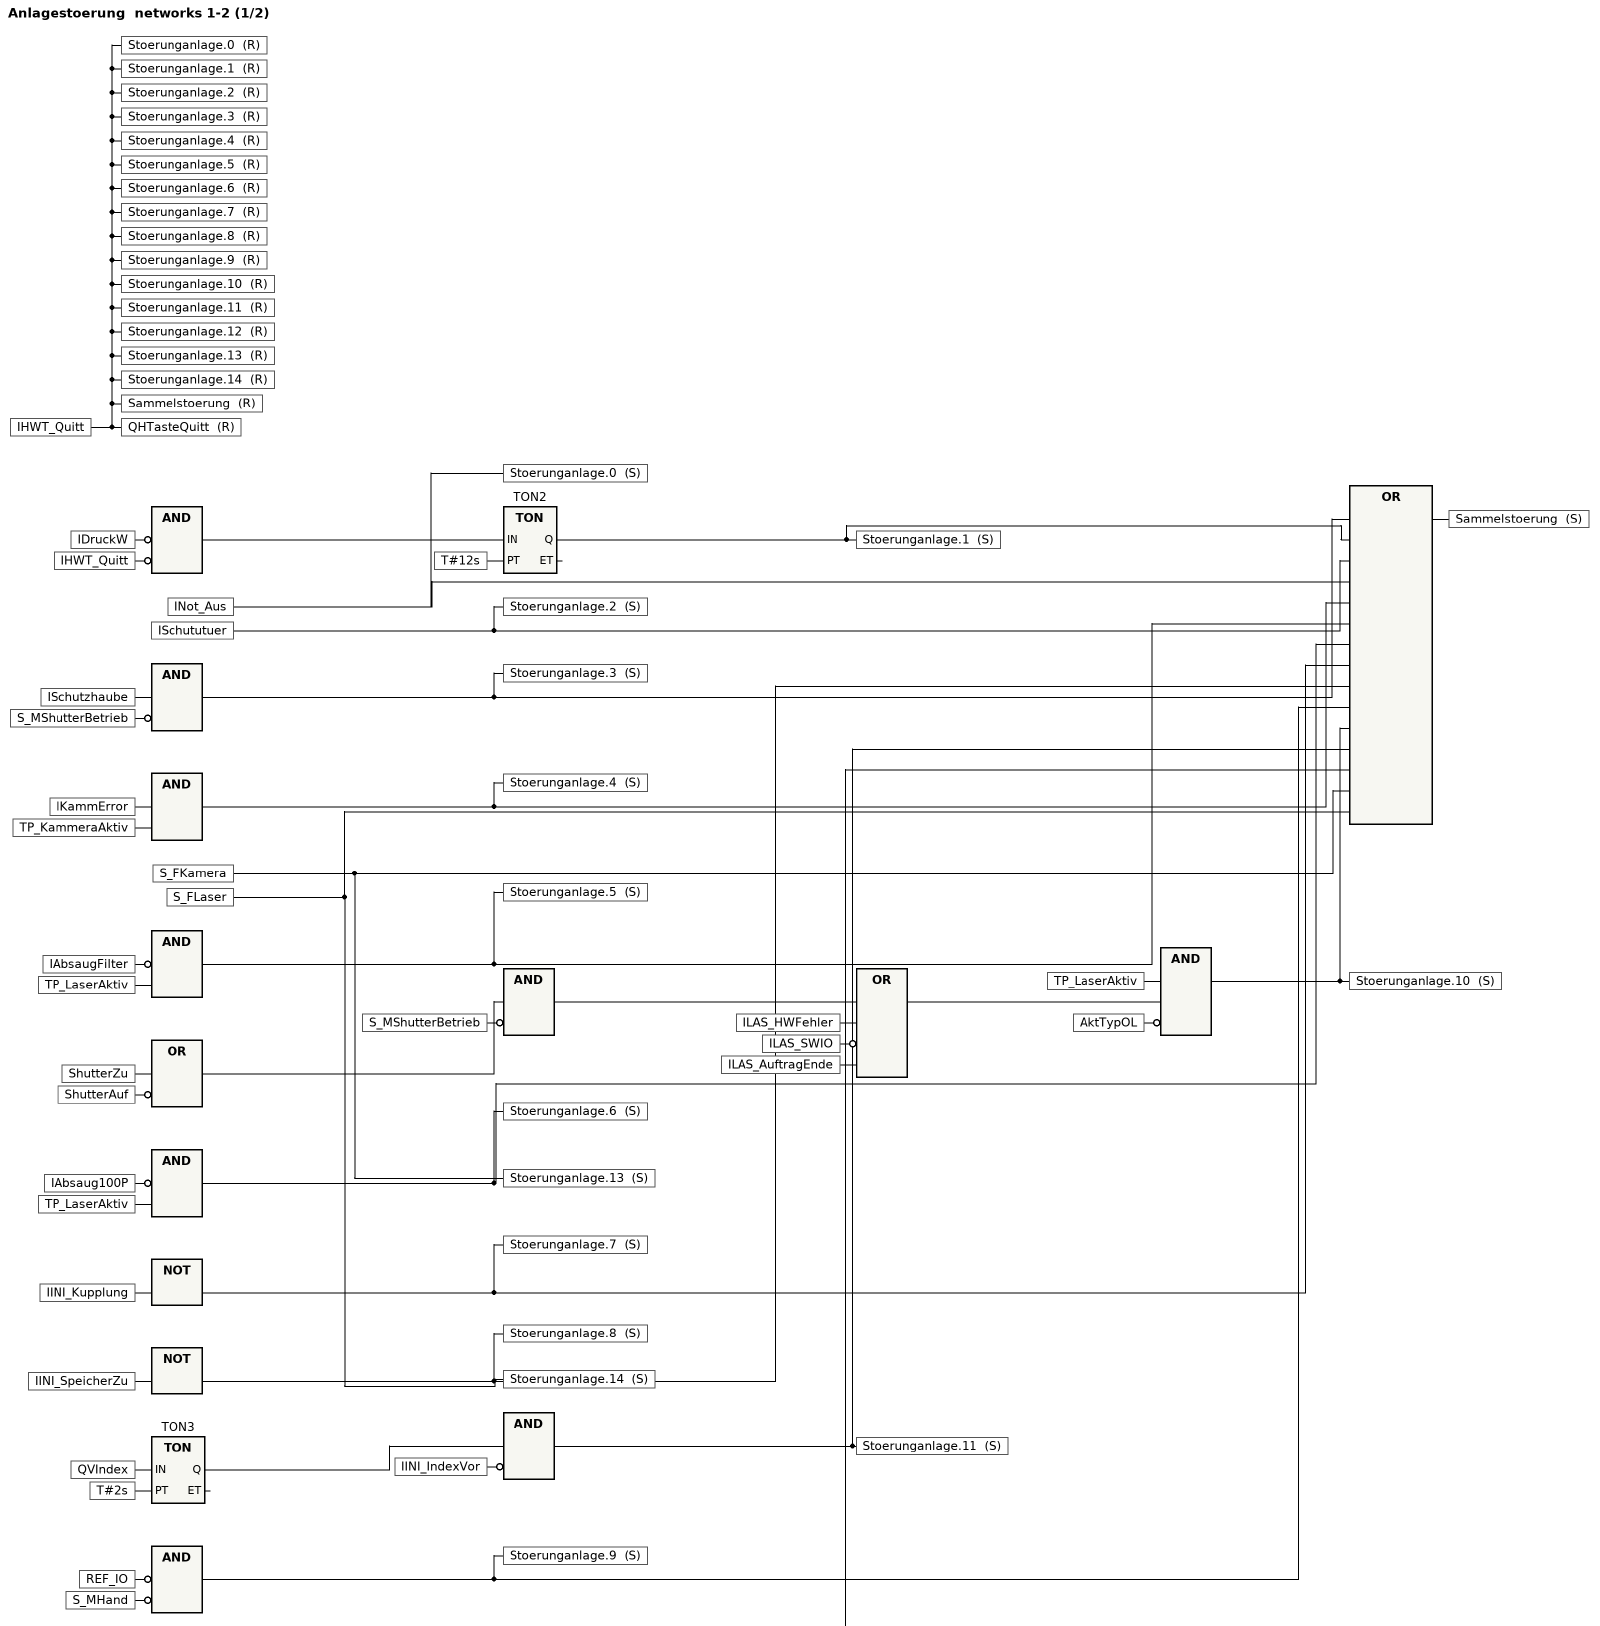
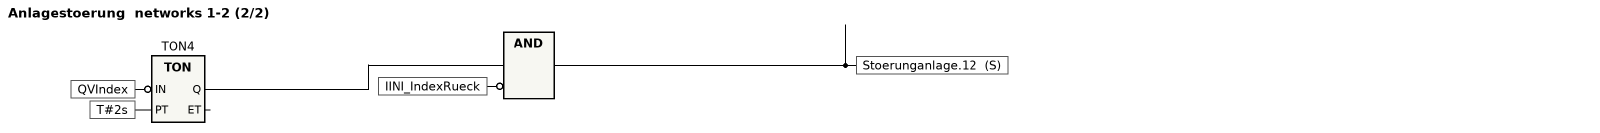
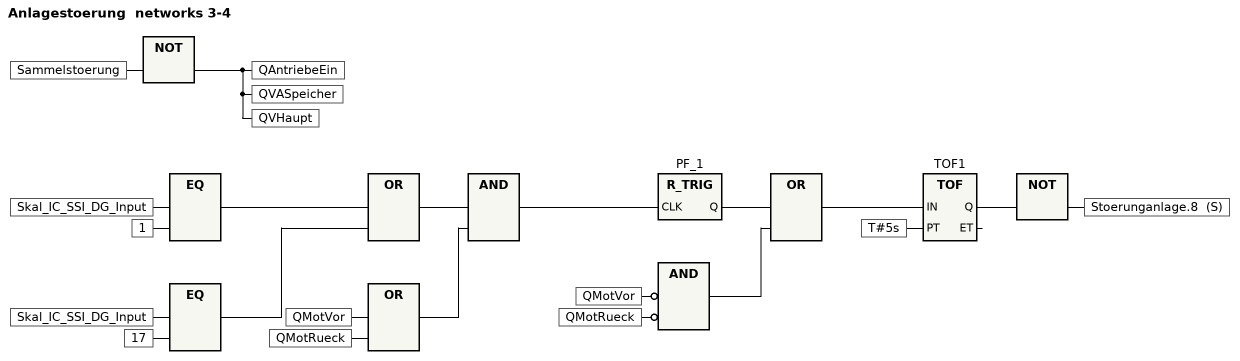
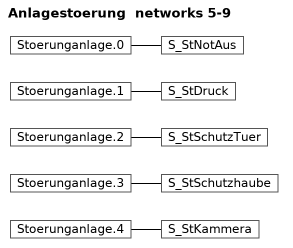
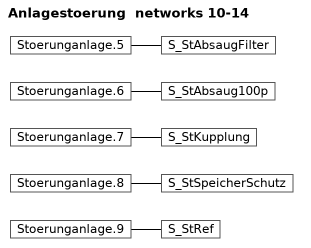
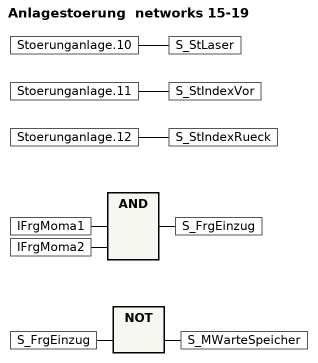
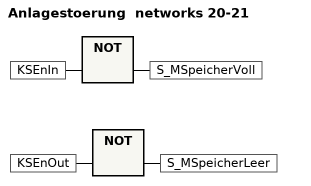
_FBD_ (* Function Block Diagram *)
NETWORK 1
	IHWT_Quitt => R Stoerunganlage.0, R Stoerunganlage.1, R Stoerunganlage.2, R Stoerunganlage.3, R Stoerunganlage.4, R Stoerunganlage.5, R Stoerunganlage.6, R Stoerunganlage.7, R Stoerunganlage.8, R Stoerunganlage.9, R Stoerunganlage.10, R Stoerunganlage.11, R Stoerunganlage.12, R Stoerunganlage.13, R Stoerunganlage.14, R Sammelstoerung, R QHTasteQuitt
NETWORK 2
	OR(<INot_Aus => S Stoerunganlage.0>, <TON2:TON(IN: AND(NOT IDruckW, NOT IHWT_Quitt), PT: T#12s) => S Stoerunganlage.1>, <ISchututuer => S Stoerunganlage.2>, <AND(ISchutzhaube, NOT S_MShutterBetrieb) => S Stoerunganlage.3>, <AND(IKammError, TP_KammeraAktiv) => S Stoerunganlage.4>, <AND(NOT IAbsaugFilter, TP_LaserAktiv) => S Stoerunganlage.5>, <AND(NOT IAbsaug100P, TP_LaserAktiv) => S Stoerunganlage.6>, <NOT IINI_Kupplung => S Stoerunganlage.7>, <NOT IINI_SpeicherZu => S Stoerunganlage.8>, <AND(NOT REF_IO, NOT S_MHand) => S Stoerunganlage.9>, <AND(TP_LaserAktiv, OR(AND(OR(ShutterZu, NOT ShutterAuf), NOT S_MShutterBetrieb), ILAS_HWFehler, NOT ILAS_SWIO, ILAS_AuftragEnde), NOT AktTypOL) => S Stoerunganlage.10>, <AND(TON3:TON(IN: QVIndex, PT: T#2s), NOT IINI_IndexVor) => S Stoerunganlage.11>, <AND(TON4:TON(IN: NOT QVIndex, PT: T#2s), NOT IINI_IndexRueck) => S Stoerunganlage.12>, <S_FKamera => S Stoerunganlage.13>, <S_FLaser => S Stoerunganlage.14>) => S Sammelstoerung
NETWORK 3
	NOT Sammelstoerung => QAntriebeEin, QVASpeicher, QVHaupt
NETWORK 4
	NOT(TOF1:TOF(IN: OR(PF_1:R_TRIG(CLK: AND(OR(EQ(Skal_IC_SSI_DG_Input, 1), EQ(Skal_IC_SSI_DG_Input, 17)), OR(QMotVor, QMotRueck))), AND(NOT QMotVor, NOT QMotRueck)), PT: T#5s)) => S Stoerunganlage.8
NETWORK 5
	Stoerunganlage.0 => S_StNotAus
NETWORK 6
	Stoerunganlage.1 => S_StDruck
NETWORK 7
	Stoerunganlage.2 => S_StSchutzTuer
NETWORK 8
	Stoerunganlage.3 => S_StSchutzhaube
NETWORK 9
	Stoerunganlage.4 => S_StKammera
NETWORK 10
	Stoerunganlage.5 => S_StAbsaugFilter
NETWORK 11
	Stoerunganlage.6 => S_StAbsaug100p
NETWORK 12
	Stoerunganlage.7 => S_StKupplung
NETWORK 13
	Stoerunganlage.8 => S_StSpeicherSchutz
NETWORK 14
	Stoerunganlage.9 => S_StRef
NETWORK 15
	Stoerunganlage.10 => S_StLaser
NETWORK 16
	Stoerunganlage.11 => S_StIndexVor
NETWORK 17
	Stoerunganlage.12 => S_StIndexRueck
NETWORK 18
	AND(IFrgMoma1, IFrgMoma2) => S_FrgEinzug
NETWORK 19
	NOT S_FrgEinzug => S_MWarteSpeicher
NETWORK 20
	NOT KSEnIn => S_MSpeicherVoll
NETWORK 21
	NOT KSEnOut => S_MSpeicherLeer
_END_FBD_
(* the same logic as Structured Text *)
(* Network 1 *)
IF IHWT_Quitt THEN Stoerunganlage.0 := FALSE; Stoerunganlage.1 := FALSE; Stoerunganlage.2 := FALSE; Stoerunganlage.3 := FALSE; Stoerunganlage.4 := FALSE; Stoerunganlage.5 := FALSE; Stoerunganlage.6 := FALSE; Stoerunganlage.7 := FALSE; Stoerunganlage.8 := FALSE; Stoerunganlage.9 := FALSE; Stoerunganlage.10 := FALSE; Stoerunganlage.11 := FALSE; Stoerunganlage.12 := FALSE; Stoerunganlage.13 := FALSE; Stoerunganlage.14 := FALSE; Sammelstoerung := FALSE; QHTasteQuitt := FALSE; END_IF;
(* Network 2 *)
IF INot_Aus THEN Stoerunganlage.0 := TRUE; END_IF;
TON2(IN := NOT IDruckW AND NOT IHWT_Quitt, PT := T#12s);
IF TON2.Q THEN Stoerunganlage.1 := TRUE; END_IF;
IF ISchututuer THEN Stoerunganlage.2 := TRUE; END_IF;
IF ISchutzhaube AND NOT S_MShutterBetrieb THEN Stoerunganlage.3 := TRUE; END_IF;
IF IKammError AND TP_KammeraAktiv THEN Stoerunganlage.4 := TRUE; END_IF;
IF NOT IAbsaugFilter AND TP_LaserAktiv THEN Stoerunganlage.5 := TRUE; END_IF;
IF NOT IAbsaug100P AND TP_LaserAktiv THEN Stoerunganlage.6 := TRUE; END_IF;
IF NOT IINI_Kupplung THEN Stoerunganlage.7 := TRUE; END_IF;
IF NOT IINI_SpeicherZu THEN Stoerunganlage.8 := TRUE; END_IF;
IF NOT REF_IO AND NOT S_MHand THEN Stoerunganlage.9 := TRUE; END_IF;
IF TP_LaserAktiv AND (((ShutterZu OR NOT ShutterAuf) AND NOT S_MShutterBetrieb) OR ILAS_HWFehler OR NOT ILAS_SWIO OR ILAS_AuftragEnde) AND NOT AktTypOL THEN Stoerunganlage.10 := TRUE; END_IF;
TON3(IN := QVIndex, PT := T#2s);
IF TON3.Q AND NOT IINI_IndexVor THEN Stoerunganlage.11 := TRUE; END_IF;
TON4(IN := NOT QVIndex, PT := T#2s);
IF TON4.Q AND NOT IINI_IndexRueck THEN Stoerunganlage.12 := TRUE; END_IF;
IF S_FKamera THEN Stoerunganlage.13 := TRUE; END_IF;
IF S_FLaser THEN Stoerunganlage.14 := TRUE; END_IF;
IF INot_Aus OR TON2.Q OR ISchututuer OR (ISchutzhaube AND NOT S_MShutterBetrieb) OR (IKammError AND TP_KammeraAktiv) OR (NOT IAbsaugFilter AND TP_LaserAktiv) OR (NOT IAbsaug100P AND TP_LaserAktiv) OR NOT IINI_Kupplung OR NOT IINI_SpeicherZu OR (NOT REF_IO AND NOT S_MHand) OR (TP_LaserAktiv AND (((ShutterZu OR NOT ShutterAuf) AND NOT S_MShutterBetrieb) OR ILAS_HWFehler OR NOT ILAS_SWIO OR ILAS_AuftragEnde) AND NOT AktTypOL) OR (TON3.Q AND NOT IINI_IndexVor) OR (TON4.Q AND NOT IINI_IndexRueck) OR S_FKamera OR S_FLaser THEN Sammelstoerung := TRUE; END_IF;
(* Network 3 *)
QAntriebeEin := NOT Sammelstoerung;
QVASpeicher := QAntriebeEin;
QVHaupt := QAntriebeEin;
(* Network 4 *)
PF_1(CLK := ((Skal_IC_SSI_DG_Input = 1) OR (Skal_IC_SSI_DG_Input = 17)) AND (QMotVor OR QMotRueck));
TOF1(IN := PF_1.Q OR (NOT QMotVor AND NOT QMotRueck), PT := T#5s);
IF NOT TOF1.Q THEN Stoerunganlage.8 := TRUE; END_IF;
(* Network 5 *)
S_StNotAus := Stoerunganlage.0;
(* Network 6 *)
S_StDruck := Stoerunganlage.1;
(* Network 7 *)
S_StSchutzTuer := Stoerunganlage.2;
(* Network 8 *)
S_StSchutzhaube := Stoerunganlage.3;
(* Network 9 *)
S_StKammera := Stoerunganlage.4;
(* Network 10 *)
S_StAbsaugFilter := Stoerunganlage.5;
(* Network 11 *)
S_StAbsaug100p := Stoerunganlage.6;
(* Network 12 *)
S_StKupplung := Stoerunganlage.7;
(* Network 13 *)
S_StSpeicherSchutz := Stoerunganlage.8;
(* Network 14 *)
S_StRef := Stoerunganlage.9;
(* Network 15 *)
S_StLaser := Stoerunganlage.10;
(* Network 16 *)
S_StIndexVor := Stoerunganlage.11;
(* Network 17 *)
S_StIndexRueck := Stoerunganlage.12;
(* Network 18 *)
S_FrgEinzug := IFrgMoma1 AND IFrgMoma2;
(* Network 19 *)
S_MWarteSpeicher := NOT S_FrgEinzug;
(* Network 20 *)
S_MSpeicherVoll := NOT KSEnIn;
(* Network 21 *)
S_MSpeicherLeer := NOT KSEnOut;
END_FUNCTION_BLOCK

(* POU Funktionsbausteine/Lasersteuerung, FBD *)
FUNCTION_BLOCK Lasersteuerung
VAR_INPUT
END_VAR
VAR_OUTPUT
END_VAR
VAR
	RS1: RS;
	PF_1: R_TRIG;
	PF_2: R_TRIG;
	NF_2: F_TRIG;
	TON1: TON;
	SR1: SR;
	PF3: R_TRIG;
	RS2: RS;
	PF4: R_TRIG;
	TP1: TP;
	NF_1: F_TRIG;
END_VAR
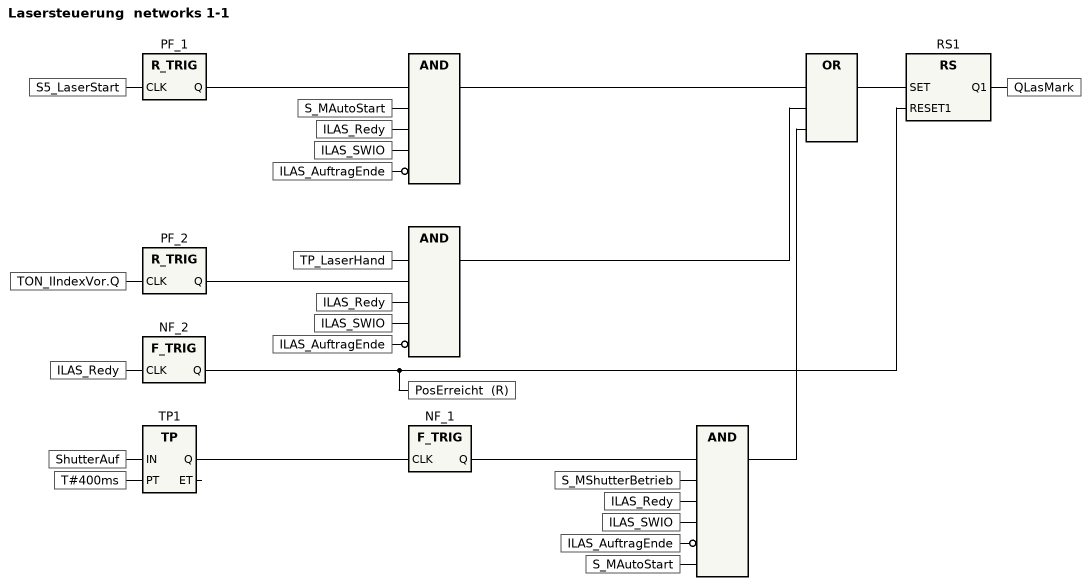
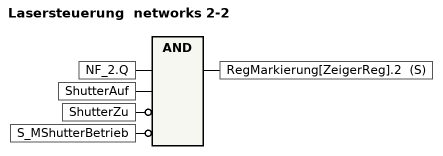
_FBD_ (* Function Block Diagram *)
NETWORK 1
	RS1:RS(SET: OR(AND(PF_1:R_TRIG(CLK: S5_LaserStart), S_MAutoStart, ILAS_Redy, ILAS_SWIO, NOT ILAS_AuftragEnde), AND(TP_LaserHand, PF_2:R_TRIG(CLK: TON_IIndexVor.Q), ILAS_Redy, ILAS_SWIO, NOT ILAS_AuftragEnde), AND(NF_1:F_TRIG(CLK: TP1:TP(IN: ShutterAuf, PT: T#400ms)), S_MShutterBetrieb, ILAS_Redy, ILAS_SWIO, NOT ILAS_AuftragEnde, S_MAutoStart)), RESET1: <NF_2:F_TRIG(CLK: ILAS_Redy) => R PosErreicht>) => QLasMark
NETWORK 2
	AND(NF_2.Q, ShutterAuf, NOT ShutterZu, NOT S_MShutterBetrieb) => S RegMarkierung[ZeigerReg].2
_END_FBD_
(* the same logic as Structured Text *)
(* Network 1 *)
PF_1(CLK := S5_LaserStart);
PF_2(CLK := TON_IIndexVor.Q);
TP1(IN := ShutterAuf, PT := T#400ms);
NF_1(CLK := TP1.Q);
NF_2(CLK := ILAS_Redy);
IF NF_2.Q THEN PosErreicht := FALSE; END_IF;
RS1(SET := (PF_1.Q AND S_MAutoStart AND ILAS_Redy AND ILAS_SWIO AND NOT ILAS_AuftragEnde) OR (TP_LaserHand AND PF_2.Q AND ILAS_Redy AND ILAS_SWIO AND NOT ILAS_AuftragEnde) OR (NF_1.Q AND S_MShutterBetrieb AND ILAS_Redy AND ILAS_SWIO AND NOT ILAS_AuftragEnde AND S_MAutoStart), RESET1 := NF_2.Q);
QLasMark := RS1.Q1;
(* Network 2 *)
IF NF_2.Q AND ShutterAuf AND NOT ShutterZu AND NOT S_MShutterBetrieb THEN RegMarkierung[ZeigerReg].2 := TRUE; END_IF;
END_FUNCTION_BLOCK

(* POU Funktionsbausteine/LaserMeldungKontrolle, ST *)
FUNCTION_BLOCK LaserMeldungKontrolle
VAR_INPUT
	Quitt_Fehler:BOOL;
	Kontrolle_Aktiv:BOOL;
END_VAR


VAR CONSTANT
	Offset_LMKontrolle: INT:=20;
END_VAR
Zeiger_LMKontrolle:=Zeiger_LMKontrolle-Offset_LMKontrolle;

IF Zeiger_LMKontrolle<1  THEN
	Zeiger_LMKontrolle:=Zeiger_LMKontrolle-Offset_LMKontrolle+500;
END_IF



(* Bearbeitung nur wenn Trigger nächstes Glied und Eintrag Gültig *)
IF	ImpulsPos=TRUE THEN
	IF RegMarkierung[Zeiger_LMKontrolle].1=TRUE AND RegMarkierung[Zeiger_LMKontrolle].2= FALSE THEN
	 	RegMarkierung[Zeiger_LMKontrolle].3:= TRUE;
		FNichtMarkiert:=TRUE;
	END_IF
END_IF
IF Quitt_Fehler = TRUE THEN
	FNichtMarkiert:=FALSE;
END_IF
END_FUNCTION_BLOCK

(* POU Funktionsbausteine/Kammera, ST *)
FUNCTION_BLOCK Kammera
VAR_INPUT
END_VAR
VAR_OUTPUT
	FehlerKammera: BOOL;
	FehlerLaser: BOOL;
	VQKammTrigg: BOOL;
END_VAR
VAR
	Zeiger_Kammera:INT;
	V1: BOOL;
	Zeiger_Kammera2: INT;
END_VAR
VAR CONSTANT
	Offset_Pos_Kammera: INT := 60;
	Offset_Pos_Kammera2: INT:= 61;
END_VAR
(* Zeiger auf Glied unter Kammera*)
Zeiger_Kammera:=ZeigerReg-Offset_Pos_Kammera;
IF	Zeiger_Kammera < 1 THEN
	Zeiger_Kammera:=ZeigerReg-Offset_Pos_Kammera+500;
END_IF

(* Zeiger auf Glied hinter  Kammera*)
Zeiger_Kammera2:=ZeigerReg-Offset_Pos_Kammera2;
IF	Zeiger_Kammera2 < 1 THEN
	Zeiger_Kammera2:=ZeigerReg-Offset_Pos_Kammera2+500;
END_IF

(* Bearbeitung nur bei Glied Anfang *)
IF  ImpulsPos = TRUE THEN
	(*  Wenn im Register Lasersollstelle eingetragen dann Triggerimpuls bilden *)
	IF  RegMarkierung[Zeiger_Kammera].1 = TRUE THEN
		VQKammTrigg:= TRUE;
	ELSE
		VQKammTrigg:= FALSE;
	END_IF
END_IF

(* Wenn Kammera Muster erkennt dann in Register eintragen *)
IF  VQKammTrigg = TRUE AND IKammOutput = TRUE THEN
	RegMarkierung[Zeiger_Kammera].4 := TRUE;
END_IF

(* Auswerten *)
(* Wenn hinter Kammera im Register Laserstelle eingetragen und kein Eintrag von der Kammera dann Fehler ausgeben *)
(*Zähler Kammera hat Fehler Erkannt hochzählen*)

IF   ImpulsPos = TRUE THEN
	IF RegMarkierung[Zeiger_Kammera2].1= TRUE AND RegMarkierung[Zeiger_Kammera2].4 = FALSE AND TP_KammeraAktiv = TRUE THEN
		FehlerKammera:=TRUE;
		SI_FKamera:=SI_FKamera+1;
	END_IF
END_IF

IF   ImpulsPos = TRUE  THEN
	IF RegMarkierung[Zeiger_Kammera2].1= TRUE AND RegMarkierung[Zeiger_Kammera2].2 = FALSE THEN
		FehlerLaser:=TRUE;
		SI_FLaser:=SI_FLaser+1;
	END_IF
END_IF


IF   ImpulsPos = TRUE THEN
	IF (RegMarkierung[Zeiger_Kammera2].1= TRUE AND RegMarkierung[Zeiger_Kammera2].2 = FALSE) OR  (RegMarkierung[Zeiger_Kammera2].1= TRUE AND RegMarkierung[Zeiger_Kammera2].4 = FALSE)THEN
	SI_NIO:=SI_NIO+1;
	END_IF
END_IF

IF   ImpulsPos = TRUE THEN
	IF RegMarkierung[Zeiger_Kammera2].1= TRUE AND RegMarkierung[Zeiger_Kammera2].2 = TRUE AND RegMarkierung[Zeiger_Kammera2].4 = TRUE THEN
	SI_IO:=SI_IO+1;
	END_IF
END_IF

IF	IHWT_Quitt = TRUE THEN
	FehlerKammera:=FALSE;
	FehlerLaser:=FALSE;
END_IF
END_FUNCTION_BLOCK

(* POU Nockenschaltwerk, ST *)
PROGRAM Nockenschaltwerk
VAR
	Zeiger :INT:=0;
	Nocke:BOOL:=FALSE;
	Zaeler:WORD;
	(*Skal_IC_SSI_DG_Input: DINT;*)
	Skal_IC_SSI_DG_Input_Alt:DINT;
	Skal_IC_SSI_DG_Input_Delta:DINT;
	Skal_SSI_DG_4_Alt: DINT;
	ImpulsPos4: BOOL;
END_VAR
(*  Miroslav Knezevic TCM 19.03.07  *)
(* Baustein bildet Zeiger für Speicher (Speichertiefe 500 Glieder) und Zeiger für Kette ( Speichertiefe variabel*)
(* Baustein liefert Impulse bei drehen in positiver Richtung und impulse bei Drehen in negativer Richtung*)
(*  Das Nockenschaltwerk liefert 32 Impulse (32 Glieder(Zähne)  bei einer Umdrehung des SSI Drehgebers *)
(* Voller Kreis = 16777216 Inkremente,  1 Impuls= 524288 Inkremente *)



Skal_IC_SSI_DG_Input:=IASSIDgInput/524288;
Skal_IC_SSI_DG_Input_Delta:=Skal_IC_SSI_DG_Input - Skal_IC_SSI_DG_Input_Alt;


(* Bildung der Viertelgliedimpulse *)
Skal_SSI_DG_4:=IASSIDgInput/131072;
IF Skal_SSI_DG_4 <> Skal_SSI_DG_4_Alt THEN
	ImpulsPos4:=TRUE;
ELSE
	ImpulsPos4:=FALSE;
END_IF
Skal_SSI_DG_4_Alt:=Skal_SSI_DG_4;


IF Skal_IC_SSI_DG_Input_Delta<-10 THEN
	Skal_IC_SSI_DG_Input_Delta:=1;
END_IF

IF Skal_IC_SSI_DG_Input_Delta>10 THEN
	Skal_IC_SSI_DG_Input_Delta:=-1;
END_IF


ZeigerReg:=DINT_TO_INT(ZeigerReg+Skal_IC_SSI_DG_Input_Delta);
IF ZeigerReg>500 THEN
	ZeigerReg:=ZeigerReg-500;
END_IF
IF ZeigerReg<1 THEN
	ZeigerReg:=ZeigerReg+500;
END_IF


ZeigerKette:=DINT_TO_INT(ZeigerKette+Skal_IC_SSI_DG_Input_Delta);
IF ZeigerKette>KettenTyp[AktTypindex,0] THEN
	ZeigerKette:=ZeigerKette-KettenTyp[AktTypindex,0];
END_IF

IF ZeigerKette<1 THEN
	ZeigerKette:=ZeigerKette+KettenTyp[AktTypindex,0];
END_IF


IF Skal_IC_SSI_DG_Input_Delta>0 THEN
	ImpulsPos:=TRUE;
ELSE
	ImpulsPos:=FALSE;
END_IF;

IF Skal_IC_SSI_DG_Input_Delta<0 THEN
	ImpulsNeg:=TRUE;
ELSE
	ImpulsNeg:=FALSE;
END_IF;



Skal_IC_SSI_DG_Input_Alt:=Skal_IC_SSI_DG_Input;
END_PROGRAM

(* POU Schrittkette, SFC *)
PROGRAM Schrittkette
VAR
END_VAR
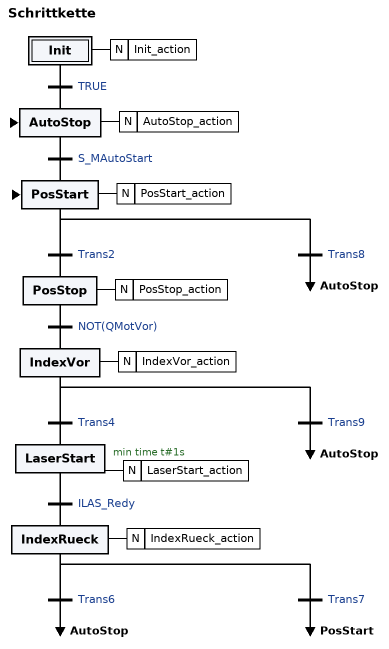
INITIAL_STEP Init:
	Init_action(N);
END_STEP
TRANSITION FROM Init TO AutoStop := TRUE;
END_TRANSITION
STEP AutoStop:
	AutoStop_action(N);
END_STEP
TRANSITION FROM AutoStop TO PosStart := S_MAutoStart;
END_TRANSITION
STEP PosStart:
	PosStart_action(N);
END_STEP
TRANSITION FROM PosStart TO PosStop := Trans2;
END_TRANSITION
TRANSITION FROM PosStart TO AutoStop := Trans8;
END_TRANSITION
STEP PosStop:
	PosStop_action(N);
END_STEP
TRANSITION FROM PosStop TO IndexVor := NOT(QMotVor);
END_TRANSITION
STEP IndexVor:
	IndexVor_action(N);
END_STEP
TRANSITION FROM IndexVor TO LaserStart := Trans4;
END_TRANSITION
TRANSITION FROM IndexVor TO AutoStop := Trans9;
END_TRANSITION
STEP LaserStart: (* min time t#1s *)
	LaserStart_action(N);
END_STEP
TRANSITION FROM LaserStart TO IndexRueck := ILAS_Redy;
END_TRANSITION
STEP IndexRueck:
	IndexRueck_action(N);
END_STEP
TRANSITION FROM IndexRueck TO AutoStop := Trans6;
END_TRANSITION
TRANSITION FROM IndexRueck TO PosStart := Trans7;
END_TRANSITION

ACTION Init_action:
_FBD_ (* Function Block Diagram *)
_END_FBD_
END_ACTION

ACTION AutoStop_action:
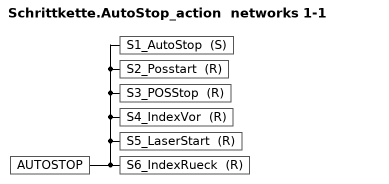
_FBD_ (* Function Block Diagram *)
NETWORK 1
	AUTOSTOP => S S1_AutoStop, R S2_Posstart, R S3_POSStop, R S4_IndexVor, R S5_LaserStart, R S6_IndexRueck
_END_FBD_
(* the same logic as Structured Text *)
(* Network 1 *)
IF AUTOSTOP THEN S1_AutoStop := TRUE; S2_Posstart := FALSE; S3_POSStop := FALSE; S4_IndexVor := FALSE; S5_LaserStart := FALSE; S6_IndexRueck := FALSE; END_IF;
END_ACTION

ACTION PosStart_action:
